INTERFACE I_Mediator

METHOD notify : BOOL
VAR_INPUT
	in_sSenderName		: STRING;
	in_sEvent 			: STRING;
END_VAR
END_METHOD

END_INTERFACE

(* stored: Version 1.1.0.1
   Itf I_Mediator: Id {55a43a09-4e5b-4a54-954c-59d6c7989341}
   Method notify: Id {1d52a1be-78d9-4edc-a3a8-0ae370d161be} *)
